ABB RAPID module: 0071DA77

MODULE ObelixMov
    !***********************************************************
    !
    ! Module:  ObelixMov
    !
    ! Description:
    !   Move the robot
    !
    ! Author: pol & victor
    !
    ! Version: 0.1.0
    !
    !***********************************************************

    CONST robtarget pHome    :=[[507.9,-6.43,715.02],[0.697685,-0.00154316,0.716328,-0.0103435],[-1,-1,-1,0],[9E+09,9E+09,9E+09,9E+09,9E+09,9E+09]];
	CONST robtarget pConvRef :=[[-115.85074989,-570.588098876,463.263482769],[0.021373544,0.101609161,0.8695055,-0.482886048],[-2,0,-2,0],[9E+09,9E+09,9E+09,9E+09,9E+09,9E+09]];
	CONST robtarget pManRef  :=[[580,42.299990184,552.739936658],[0.51893094,-0.131239024,0.843441139,-0.045760712],[0,-1,-1,0],[9E+09,9E+09,9E+09,9E+09,9E+09,9E+09]];
	!CONST robtarget pOvenRef :=[[-400.60,632.71,501.69],[0.350259,-0.742904,0.298477,0.486132],[1,-1,-1,0],[9E+09,9E+09,9E+09,9E+09,9E+09,9E+09]];
    CONST robtarget pOvenRef :=[[-291.029880742,659.908842444,594.297264732],[0.363486279,-0.625201176,0.407577419,0.55756781],[1,0,-1,0],[9E+09,9E+09,9E+09,9E+09,9E+09,9E+09]];

    CONST num convSecOffset{3} := [0, 0, -100];   !security offset [x, y, z]
    CONST num manSecOffset{3} := [0, 0, -100];    !security offset [x, y, z]
    CONST num ovenSecOffset{3} := [0, 100, 0];   !security offset [x, y, z]

    CONST num convOffset{3} := [0, -200, 0];        !offset between 2 conv [x, y, z]
    CONST num ovenMatOffset{3} := [100, 0, -100]; !offset between oven positions [x, y, z]


    ! Points variables preallocation
    VAR robtarget pConv{2,2};
    VAR robtarget pOven{2,3,3};
    VAR robtarget pMan{2};
    CONST robtarget pHome_2:=[[507.9,-6.43,715.02],[0.697685,-0.00154316,0.716328,-0.0103435],[-1,-1,-1,0],[9E+09,9E+09,9E+09,9E+09,9E+09,9E+09]];


    !***********************************************************
    !
    ! Procedure main
    !
    !   This is the entry point of your program
    !
    !***********************************************************
    PROC main()
        TPWrite "Hello ABB";
        MoveJ pHome, v1000, fine, tool0;
        !-----------------------------------

        ! 0. Points definition
        pMan := [pManRef, Offs(pManRef, manSecOffset{1}, manSecOffset{2}, manSecOffset{3})];
        defineConvPts pConvRef, convOffset, convSecOffset, pConv;
        defineOvenPts pOvenRef, ovenMatOffset, ovenSecOffset, pOven;

        man2conv pMan, pConv, 2;
        ! TEST. Movement Tests
        movTest pConv, pOven, pMan;

        !TODO: See if the mov. sequences can be extracted to a PROC (they are a sequence of MoveJ, MoveJ, MoveJ)

        !-----------------------------------
        MoveJ pHome, v1000, fine, tool0;
    ENDPROC

    !***********************************************************
    PROC defineOvenPts(robtarget orig, num matOffs{*}, num secOffs{*}, INOUT robtarget pts{*,*,*})

        !define the security points {1} and the inside oven points {2}
        FOR i FROM 1 TO 3 DO
            FOR j FROM 1 TO 3 DO
                pts{1,i,j} := Offs(orig, matOffs{1}*(i-1), matOffs{2}, matOffs{3}*(j-1));
                pts{2,i,j} := Offs(pts{1,i,j}, secOffs{1}, secOffs{2}, secOffs{3});
            ENDFOR
        ENDFOR
    ENDPROC

    !***********************************************************
    PROC defineConvPts(robtarget orig, num convOffs{*}, num secOffs{*}, INOUT robtarget pts{*,*})

        !define the security points {1} and the conv points {2}
        FOR i FROM 1 TO 2 DO
                pts{1,i} := Offs(orig, convOffs{1}*(i-1), convOffs{2}*(i-1), convOffs{3}*(i-1));
                pts{2,i} := Offs(pts{1,i}, secOffs{1}, secOffs{2}, secOffs{3});
        ENDFOR
    ENDPROC

    !***********************************************************
    PROC gotoOvenPts(robtarget pts{*,*,*})
        FOR i FROM 1 TO 3 DO
            FOR j FROM 1 TO 3 DO
                MoveJ pts{1,i,j}, v1000, fine, tool0;
                MoveJ pts{2,i,j}, v200, fine, tool0;
                MoveJ pts{1,i,j}, v200, fine, tool0;
            ENDFOR
        ENDFOR
    ENDPROC

    !***********************************************************
    PROC conv2oven(robtarget pConv{*,*}, robtarget pOven{*,*,*}, num iConv, num iOven, num jOven)

        MoveJ pConv{1, iConv}, v1000, fine, tool0;
        MoveJ pConv{2, iConv}, v200, fine, tool0;
        MoveJ pConv{1, iConv}, v200, fine, tool0;

        MoveJ pOven{1, iOven, jOven}, v1000, fine, tool0;
        MoveJ pOven{2, iOven, jOven}, v200, fine, tool0;
        MoveJ pOven{1, iOven, jOven}, v200, fine, tool0;

        !TODO: set timer taking into account iOven, jOven, chocoType
        !TODO: return to pHome?

    ENDPROC

    !***********************************************************
    PROC oven2man(robtarget pOven{*,*,*}, robtarget pMan{*}, num iOven, num jOven)

        MoveJ pOven{1, iOven, jOven}, v1000, fine, tool0;
        MoveJ pOven{2, iOven, jOven}, v200, fine, tool0;
        MoveJ pOven{1, iOven, jOven}, v200, fine, tool0;

        MoveJ pMan{1}, v1000, fine, tool0;
        MoveJ pMan{2}, v200, fine, tool0;
        MoveJ pMan{1}, v200, fine, tool0;

        !TODO: set timer for the dryer or wait 5 sections (Idle time)
        !TODO: return to pHome?

    ENDPROC

    PROC man2conv(robtarget pMan{*}, robtarget pConv{*,*}, num iConv)

        MoveJ pMan{1}, v1000, fine, tool0;
        MoveJ pMan{2}, v200, fine, tool0;
        MoveJ pMan{1}, v200, fine, tool0;

        MoveJ pConv{1, iConv}, v1000, fine, tool0;
        MoveJ pConv{2, iConv}, v200, fine, tool0;
        MoveJ pConv{1, iConv}, v200, fine, tool0;

        !TODO: set timer for the dryer or wait 5 sections (Idle time)
        !TODO: return to pHome?

    ENDPROC
    !***********************************************************
    PROC movTest(robtarget pConv{*,*}, robtarget pOven{*,*,*}, robtarget pMan{*})
        ! Perform diferent movement tests
        !oven2oven
        gotoOvenPts pOven;

        !conv2oven
        FOR i FROM 1 TO 3 DO
            FOR j FROM 1 TO 3 DO
                conv2oven pConv, pOven, 1, i, j;
            ENDFOR
        ENDFOR

        !oven2man
        FOR i FROM 1 TO 3 DO
            FOR j FROM 1 TO 3 DO
                oven2man pOven, pMan, i, j;
            ENDFOR
        ENDFOR

        !oven2home
        FOR i FROM 1 TO 3 DO
            FOR j FROM 1 TO 3 DO
                MoveJ pOven{1, i, j}, v1000, fine, tool0;
                MoveJ pHome, v1000, fine, tool0;
            ENDFOR
        ENDFOR

        !conv2home
        FOR i FROM 1 TO 2 DO
            MoveJ pConv{1, i}, v1000, fine, tool0;
            MoveJ pHome, v1000, fine, tool0;
        ENDFOR

        !man2home
        MoveJ pMan{1}, v1000, fine, tool0;
        MoveJ pHome, v1000, fine, tool0;
    ENDPROC

ENDMODULE
